SUBAPPLICATION Uebung_019 (* Umschalten einer Maske *)
  (* Standard: 61499-2; Description: Copyright (c) 2023 Meisterschulen am Ostbahnhof This program and the accompanying materials are made available under the terms of the Eclipse Public License 2.0 which is available at https://www.eclipse.org/legal/epl-2.0/ SPDX-License-Identifier: EPL-2.0 *)
  (* Version 1.0, 2023-10-23, Franz Höpfinger, Meisterschulen am Ostbahnhof *)
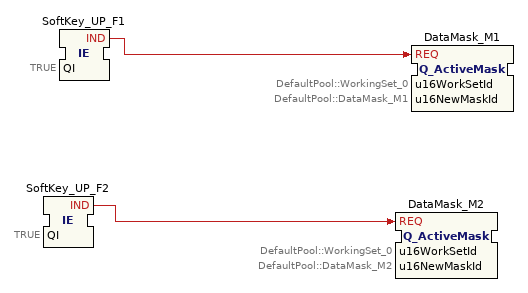
  FBS
    SoftKey_UP_F1 : IE(QI := TRUE);
    DataMask_M1 : Q_ActiveMask(u16WorkSetId := DefaultPool::WorkingSet_0, u16NewMaskId := DefaultPool::DataMask_M1);
    SoftKey_UP_F2 : IE(QI := TRUE);
    DataMask_M2 : Q_ActiveMask(u16WorkSetId := DefaultPool::WorkingSet_0, u16NewMaskId := DefaultPool::DataMask_M2);
  END_FBS
  EVENT_CONNECTIONS
    SoftKey_UP_F1.IND TO DataMask_M1.REQ;
    SoftKey_UP_F2.IND TO DataMask_M2.REQ;
  END_CONNECTIONS
END_SUBAPPLICATION
